FUNCTION_BLOCK BASIC_DLE0 (* Basic Function Block Type *)
  (* Standard: 61499-2 *)
  (* Version 0.0, 2015-11-04, 4DIAC-IDE, 4DIAC-Consortium *)
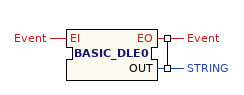
  EVENT_INPUT
    EI;
  END_EVENT
  EVENT_OUTPUT
    EO WITH OUT;
  END_EVENT
  VAR_OUTPUT
    OUT : STRING;
  END_VAR
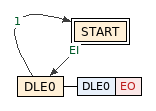
  EC_STATES
    START; (* Initial State *)
    DLE0 : DLE0 -> EO; (* Normal execution *)
  END_STATES
  EC_TRANSITIONS
    START TO DLE0 := EI;
    DLE0 TO START := 1;
  END_TRANSITIONS
  ALGORITHM DLE0 IN ST: (* Normally executed algorithm *)
OUT:='\x10\x30';
  END_ALGORITHM
END_FUNCTION_BLOCK
